// TIA Portal V20 export
TYPE "STimer"
   STRUCT
      IN : Bool;
      OUT : Bool;
      Count : Real;
      CountMax : Real;
   END_STRUCT;
END_TYPE
